Staubli VAL3: OnF1.pgx

program OnF1()
begin
  //
  if nType==1
    call setIO(sItem)
    popUpMsg("选择IO："+sItem)
  endIf

end
